{attribute 'qualified_only'}
{attribute 'strict'}
TYPE E_CX_DeviceState : (
	IDLE,
	ID,
	DEVTYPE,
	BUILDLINES,
	WRITELINE1,
	WRITELINE2,
	ERROR,
	DONE

	//E_CX_DEVICE_CX1,
	//E_CX_DEVICE_CX2
);
END_TYPE

(* stored: Version 1.1.0.1
   DUT E_CX_DeviceState: Id {1be32b35-edc1-4dbc-8f31-91317a9c14a4} *)
